{attribute 'qualified_only'}
{attribute 'strict'}
TYPE CmdMotorOnOff :
(
	None,
	Reset,
	StartFwd,
	StartRev,
	Stop	
);
END_TYPE

(* stored: Version 1.1.0.1, ProductVersion 3.1.4022.11
   DUT CmdMotorOnOff: Id {15d8907b-2bb9-4f13-b9da-e3f4d730637c} *)
